Omron CX-Programmer project NewProject (CX-Programmer 9.61)

# PLC NewPLC1: CPM2* 

## Global symbols (name address type ; comment)
0.00 BOOL  ; passo a passo formador fila entrada roler 41
DM0 CHANNEL  ; peças roller MF 41

## Program NewProgram1 (no task)
Local symbols
KEEP 30.00 BOOL
PH29paradaT1 DM1 CHANNEL  ; cnt prensa 31 parada T1
PH29paradaT2 DM4 CHANNEL  ; cnt prensa 31 parada T2
PH29paradaT3 DM7 CHANNEL  ; cnt prensa 31 parada T3
PH30paradaT1 DM2 CHANNEL  ; cnt prensa 31 parada T1
PH30paradaT2 DM5 CHANNEL  ; cnt prensa 31 parada T2
PH30paradaT3 DM8 CHANNEL  ; cnt prensa 31 parada T3
PH31paradaT1 DM3 CHANNEL  ; cnt prensa 31 parada T1
PH31paradaT2 DM6 CHANNEL  ; cnt prensa 31 parada T2
PH31paradaT3 DM9 CHANNEL  ; cnt prensa 31 parada T3
anoRelogio DM210 CHANNEL  ; Ano Relógio
codFormPH29 DM409 CHANNEL  ; Codigo do formato ph29
codFormPH30 DM407 CHANNEL  ; Codigo do formato ph30
codFormPH31 DM405 CHANNEL  ; Codigo do formato ph31
delayCicloPrensa29 TIM001 BOOL  ; Retardo ciclo da prensa
delayCicloPrensa30 TIM002 BOOL  ; Retardo ciclo da prensa
delayCicloPrensa31 TIM003 BOOL  ; Retardo ciclo da prensa
diaCalendario DM806 CHANNEL  ; dia calendario
diaMes DM400 CHANNEL  ; dia do mes
diaRelogio DM208 CHANNEL  ; Dia Relógio
filtroCntPc29 TIM021 BOOL  ; filtro contagem peças
filtroCntPc30 TIM020 BOOL  ; filtro contagem peças
filtroCntPc31 TIM023 BOOL  ; filtro contagem peças
firstDMenvioFormat DM410 CHANNEL  ; primeiro DM envio formato
firstDMenvioPcPH DM402 CHANNEL  ; pirmeiro DM de envio peças ph
horaRelogio DM207 CHANNEL  ; Horas Relogio
horas DM800 CHANNEL  ; horas
linhaSelect DM811 CHANNEL  ; linha selecionada
mesCalendario DM808 CHANNEL  ; mes calendario
mesRelogio DM209 CHANNEL  ; Mes Relogio
mesSelecionado DM810 CHANNEL  ; mês selecionado
mesSelect DM910 CHANNEL  ; mês selecionado
minutos DM802 CHANNEL  ; minutos
minutosRelogio DM206 CHANNEL  ; Minutos Relógio
numberCavidPH29 DM408 CHANNEL  ; Número cavidades na prensa29
numberCavidPH30 DM406 CHANNEL  ; Número cavidades na prensa30
numberCavidPH31 DM404 CHANNEL  ; Número cavidades na prensa31
pecaPH29 DM100 CHANNEL  ; conta peças ph29
pecaPH30 DM102 CHANNEL  ; conta peças ph30
pecaPH31 DM104 CHANNEL  ; conta peças ph31
pecaRoller41 DM106 CHANNEL  ; contagem de peças roller 41
pecaRoller42 DM108 CHANNEL  ; contagem de peças roller 42
pecaRoller43 DM110 CHANNEL  ; contagem de peças roller 43
ph29parada 20.00 BOOL  ; prensa 29 parada
ph30parada 21.00 BOOL  ; prensa 30 parada
ph31parada 22.00 BOOL  ; prensa 31 parada
prensa29 0.02 BOOL  ; Prensa 29
prensa30 0.01 BOOL  ; Prensa 30
prensa31 0.00 BOOL  ; Prensa 31
relogio4dig DM211 CHANNEL  ; Ano Relógio 4 digitos
segundos DM804 CHANNEL  ; segundos
segundosRelogio DM205 CHANNEL  ; Segundos Relógio

### Section main

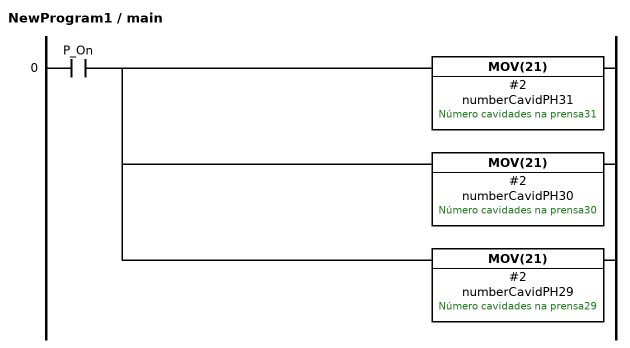
; rung 0
LD P_On
MOV(21) #2 numberCavidPH31  ; Número cavidades na prensa31
MOV(21) #2 numberCavidPH30  ; Número cavidades na prensa30
MOV(21) #2 numberCavidPH29  ; Número cavidades na prensa29

### Section PH29

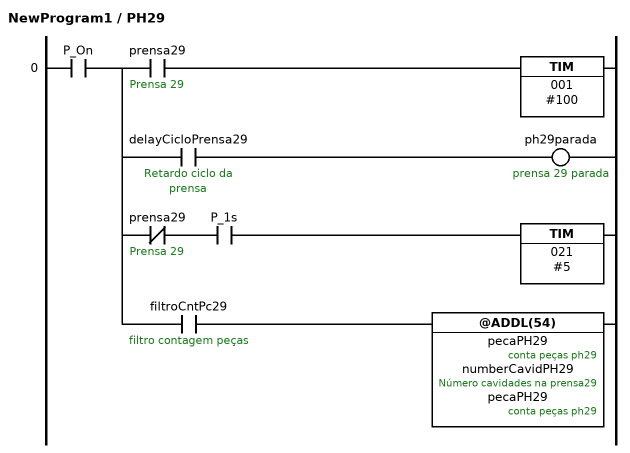
; rung 0
LD P_On
OUT TR0
AND prensa29  ; Prensa 29
TIM 001 #100
LD TR0
AND delayCicloPrensa29  ; Retardo ciclo da prensa
OUT ph29parada  ; prensa 29 parada
LD TR0
ANDNOT prensa29  ; Prensa 29
AND P_1s
TIM 021 #5
LD TR0
AND filtroCntPc29  ; filtro contagem peças
@ADDL(54) pecaPH29 numberCavidPH29 pecaPH29  ; conta peças ph29, Número cavidades na prensa29

### Section PH30

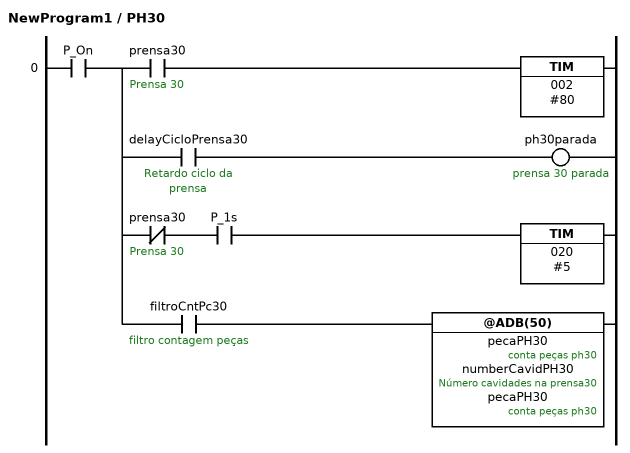
; rung 0
LD P_On
OUT TR0
AND prensa30  ; Prensa 30
TIM 002 #80
LD TR0
AND delayCicloPrensa30  ; Retardo ciclo da prensa
OUT ph30parada  ; prensa 30 parada
LD TR0
ANDNOT prensa30  ; Prensa 30
AND P_1s
TIM 020 #5
LD TR0
AND filtroCntPc30  ; filtro contagem peças
@ADB(50) pecaPH30 numberCavidPH30 pecaPH30  ; conta peças ph30, Número cavidades na prensa30

### Section PH31

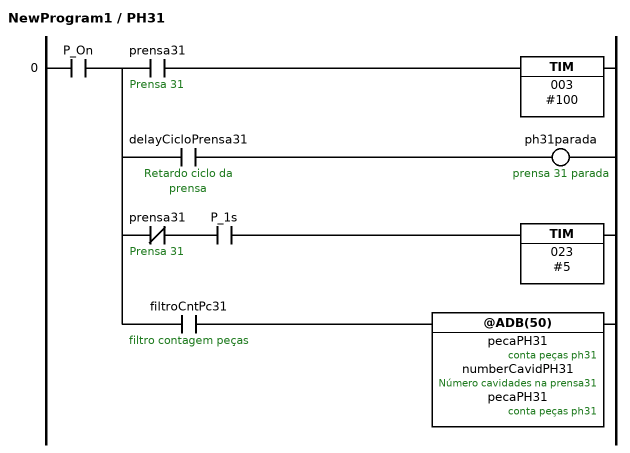
; rung 0
LD P_On
OUT TR0
AND prensa31  ; Prensa 31
TIM 003 #100
LD TR0
AND delayCicloPrensa31  ; Retardo ciclo da prensa
OUT ph31parada  ; prensa 31 parada
LD TR0
ANDNOT prensa31  ; Prensa 31
AND P_1s
TIM 023 #5
LD TR0
AND filtroCntPc31  ; filtro contagem peças
@ADB(50) pecaPH31 numberCavidPH31 pecaPH31  ; conta peças ph31, Número cavidades na prensa31

### Section Reset

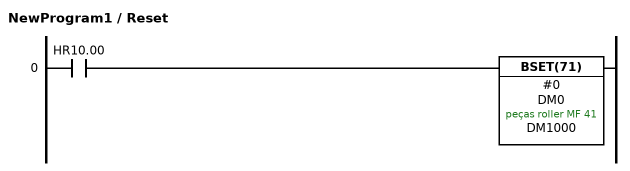
; rung 0
LD HR10.00
BSET(71) #0 DM0 DM1000  ; peças roller MF 41

### Section RollerTeste

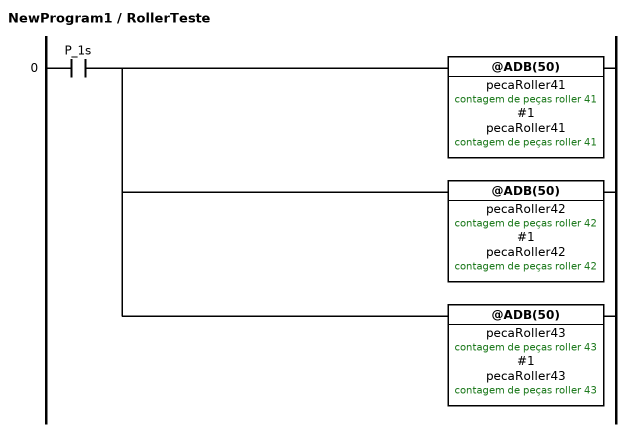
; rung 0
LD P_1s
@ADB(50) pecaRoller41 #1 pecaRoller41  ; contagem de peças roller 41
@ADB(50) pecaRoller42 #1 pecaRoller42  ; contagem de peças roller 42
@ADB(50) pecaRoller43 #1 pecaRoller43  ; contagem de peças roller 43

### Section End
; rung 0
END(01)